(* IEC 61131-3 sources: F100R_S278_Temperville/MyController.device.xml.v3^/Plc Logic.plclogic.xml.v3^/Application.application.xml.v3^/02_Operação (part 4) *)

(* ---- P_ComandosEventos.prg.st ---- *)
PROGRAM P_ComandosEventos
VAR
	TonInicioCicloEventos: ton;
	TonInicioCicloEventosIn: BOOL;
	TonInicioCicloEventosQ: BOOL;
	///------------ Disjuntores ----------------
	TpDisjGeralOn: PulsoPositivo;
	TpDisjGeralOff: PulsoPositivo;
	TpDisjResistOn: PulsoPositivo;
	TpDisjResistOff: PulsoPositivo;
	///------- Comandos Mesa de Operação -------
	TpOperacaoStandby: PulsoPositivo;
	TpOperacaoHabilitada: PulsoPositivo;
	TpBtEmergencia09On: PulsoPositivo;
	TpBtEmergencia09Off: PulsoNegativo;
	TpBt01ResetEmergencia: PulsoPositivo;
	///--- Comandos Mesa de Operação Manual ---
	TpOperacaoManual: PulsoPositivo;
	TpOperacaoAutoma: PulsoPositivo;
	TpBtEmergencia10On: PulsoPositivo;
	TpBtEmergencia10Off: PulsoNegativo;
	TpBt02ResetEmergencia: PulsoPositivo;
	///------ Comandos Mesa de Entrada ------
	TpBtEmergencia01On: PulsoPositivo;
	TpBtEmergencia01Off: PulsoNegativo;
	TpBtEmergencia02On: PulsoPositivo;
	TpBtEmergencia02Off: PulsoNegativo;
	TpBtConfirmaCarga: PulsoPositivo;
	TpChAvancoMeEntOn: PulsoPositivo;
	TpChAvancoMeEntOff: PulsoNegativo;
	TpChRecuoMeEntOn: PulsoPositivo;
	TpChRecuoMeEntOff: PulsoNegativo;
	TpGradeEntradaUp: PulsoPositivo;
	TpGradeEntradaDown: PulsoNegativo;
	TpBtEmergencia03On: PulsoPositivo;
	TpBtEmergencia03Off: PulsoNegativo;
	TpBtEmergencia04On: PulsoPositivo;
	TpBtEmergencia04Off: PulsoNegativo;
	///------ Comandos do Resfriamento ------
	TpBtEmergencia05On: PulsoPositivo;
	TpBtEmergencia05Off: PulsoNegativo;
	TpChAbreResfSup01: PulsoPositivo;
	TpChFechaResfSup01: PulsoNegativo;
	TpChAbreResfInf01: PulsoPositivo;
	TpChFechaResfInf01: PulsoNegativo;
	TpChAbreResfSup02: PulsoPositivo;
	TpChFechaResfSup02: PulsoNegativo;
	TpChAbreResfInf02: PulsoPositivo;
	TpChFechaResfInf02: PulsoNegativo;
	TpBtEmergencia06On: PulsoPositivo;
	TpBtEmergencia06Off: PulsoNegativo;
	TpChAvancoLimpVidroOn: PulsoPositivo;
	TpChAvancoLimpVidroOff: PulsoNegativo;
	TpChRecuoLimpVidroOn: PulsoPositivo;
	TpChRecuoLimpVidroOff: PulsoNegativo;
	///------- Comandos Mesa de Saida -------
	TpBtEmergencia07On: PulsoPositivo;
	TpBtEmergencia07Off: PulsoNegativo;
	TpChAvancoMeSaiOn: PulsoPositivo;
	TpChAvancoMeSaiOff: PulsoNegativo;
	TpChRecuoMeSaiOn: PulsoPositivo;
	TpChRecuoMeSaiOff: PulsoNegativo;
	TpGradeSaidaUp: PulsoPositivo;
	TpGradeSaidaDown: PulsoNegativo;
	TpBtEmergencia08On: PulsoPositivo;
	TpBtEmergencia08Off: PulsoNegativo;
	///------ Comandos do Supervisório ------
	TpBtEnvioDeReceita: PulsoPositivo;
	TpBtHmiIniciaCiclo: PulsoPositivo;
	TpBtHmiFinalizaCiclo: PulsoPositivo;
	TpBtSairForno: PulsoPositivo;
	TpBtSairResfriamento: PulsoPositivo;
	TpBtAbrePortaEntrForno: PulsoPositivo;
	TpBtFechaPortaEntForno: PulsoNegativo;
	TpBtAbrePortaSaidaForno: PulsoPositivo;
	TpBtFechaPortaSaidForno: PulsoNegativo;
	TpBtForceConveccaoOn: PulsoPositivo;
	TpBtForceConveccaoOff: PulsoNegativo;
	TpBtSobeForno: PulsoPositivo;
	TpBtDesceForno: PulsoPositivo;
	TpTesteAutoResistencia: PulsoPositivo;
	TpTesteAutoResistFim: PulsoPositivo;
	TpTesteAutoResistAbort: PulsoPositivo;
	TpProgrHorariaAtivada: PulsoPositivo;
	TpProgrHorariaDesativada: PulsoNegativo;
	TpProgrHorariaIniciadda: PulsoPositivo;
	TpBtLigaAquecimentoRampa: PulsoPositivo;
	TpBtLigaAquecimento: PulsoPositivo;
	TpBtDesligaAquecimento: PulsoPositivo;
	TpResistenciaLigada: PulsoPositivo;
	TpResistenciaDesligada: PulsoNegativo;
	TpHomeDutosIniciado: PulsoPositivo;
	TpHomeDutosOK: PulsoPositivo;
	TpHomeGuilhotinaIniciado: PulsoPositivo;
	TpHomeGuilhotinaOK: PulsoPositivo;
END_VAR

//Registro de Eventos

//Sinais Retorno Disjuntores
(*----------- Disjuntor Geral -------------*)
TpDisjGeralOn	(Entrada:= xDisjGeralOn, 	SaidaPulsoPo=> );
TpDisjGeralOff	(Entrada:= xDisjGeralOff, 	SaidaPulsoPo=> );

(*-------- Disjuntor Resistências ---------*)
TpDisjResistOn	(Entrada:= xDisjResistOn, 	SaidaPulsoPo=> );
TpDisjResistOff	(Entrada:= xDisjResistOff, 	SaidaPulsoPo=> );

//Sinais de Acionamento de Botoes Fisicos
(*------- Comandos Mesa de Operação -------*)
TpOperacaoHabilitada	(Entrada:= xOperacaoHabilitada, 	SaidaPulsoPo=> );
TpOperacaoStandby		(Entrada:= xOperacaoStandBy, 		SaidaPulsoPo=> );
TpBtEmergencia09On		(Entrada:= xBt09Emergencia, 		SaidaPulsoPo=> );
TpBtEmergencia09Off		(Entrada:= xBt09Emergencia, 		SaidaPulsoNe=> );
TpBt01ResetEmergencia	(Entrada:= xBt01CalaAlarme, 		SaidaPulsoPo=> );

(*--- Comandos Mesa de Operação Manual ---*)
TpOperacaoManual		(Entrada:= xOperacaoManual, 		SaidaPulsoPo=> );
TpOperacaoAutoma		(Entrada:= xOperacaoAutoma, 		SaidaPulsoPo=> );
TpBtEmergencia10On		(Entrada:= xBt10Emergencia,			SaidaPulsoPo=> );
TpBtEmergencia10Off		(Entrada:= xBt10Emergencia,			SaidaPulsoNe=> );
TpBt02ResetEmergencia	(Entrada:= xBt02CalaAlarme, 		SaidaPulsoPo=> );

(*------ Comandos Mesa de Entrada ------*)
TpBtEmergencia01On		(Entrada:= xBt01Emergencia,			SaidaPulsoPo=> );
TpBtEmergencia01Off		(Entrada:= xBt01Emergencia,			SaidaPulsoNe=> );
TpBtEmergencia02On		(Entrada:= xBt02Emergencia,			SaidaPulsoPo=> );
TpBtEmergencia02Off		(Entrada:= xBt02Emergencia,			SaidaPulsoNe=> );
TpBtConfirmaCarga		(Entrada:= xBtHabilitaCarregamento,	SaidaPulsoPo=> );
TpChAvancoMeEntOn		(Entrada:= xChAvancaMesaEntrada,	SaidaPulsoPo=> );
TpChAvancoMeEntOff		(Entrada:= xChAvancaMesaEntrada,	SaidaPulsoNe=> );
TpChRecuoMeEntOn		(Entrada:= xChRecuaMesaEntrada,		SaidaPulsoPo=> );
TpChRecuoMeEntOff		(Entrada:= xChRecuaMesaEntrada,		SaidaPulsoNe=> );
TpGradeEntradaUp		(Entrada:= xValvulaGradeEntrada,	SaidaPulsoPo=> );
TpGradeEntradaDown		(Entrada:= xValvulaGradeEntrada,	SaidaPulsoNe=> );
TpBtEmergencia03On		(Entrada:= xBt03Emergencia,			SaidaPulsoPo=> );
TpBtEmergencia03Off		(Entrada:= xBt03Emergencia,			SaidaPulsoNe=> );
TpBtEmergencia04On		(Entrada:= xBt04Emergencia,			SaidaPulsoPo=> );
TpBtEmergencia04Off		(Entrada:= xBt04Emergencia,			SaidaPulsoNe=> );

(*------ Comandos do Resfriamento ------*)
TpBtEmergencia05On		(Entrada:= xBt05Emergencia,			SaidaPulsoPo=> );
TpBtEmergencia05Off		(Entrada:= xBt05Emergencia,			SaidaPulsoNe=> );
TpChAbreResfSup01		(Entrada:= xChAbreDuctosResfriadorSup01,SaidaPulsoPo=> );
TpChFechaResfSup01		(Entrada:= xChAbreDuctosResfriadorSup01,SaidaPulsoNe=> );
TpChAbreResfInf01		(Entrada:= xChAbreDuctosResfriadorInf01,SaidaPulsoPo=> );
TpChFechaResfInf01		(Entrada:= xChAbreDuctosResfriadorInf01,SaidaPulsoNe=> );
TpChAbreResfSup02		(Entrada:= xChAbreDuctosResfriadorSup02,SaidaPulsoPo=> );
TpChFechaResfSup02		(Entrada:= xChAbreDuctosResfriadorSup02,SaidaPulsoNe=> );
TpChAbreResfInf02		(Entrada:= xChAbreDuctosResfriadorInf02,SaidaPulsoPo=> );
TpChFechaResfInf02		(Entrada:= xChAbreDuctosResfriadorInf02,SaidaPulsoNe=> );
TpBtEmergencia06On		(Entrada:= xBt06Emergencia,				SaidaPulsoPo=> );
TpBtEmergencia06Off		(Entrada:= xBt06Emergencia,				SaidaPulsoNe=> );
TpChAvancoLimpVidroOn	(Entrada:= xChAvancoLimpaResfriador02,	SaidaPulsoPo=> );
TpChAvancoLimpVidroOff	(Entrada:= xChAvancoLimpaResfriador02,	SaidaPulsoNe=> );
TpChRecuoLimpVidroOn	(Entrada:= xChRecuoLimpaResfriador02,	SaidaPulsoPo=> );
TpChRecuoLimpVidroOff	(Entrada:= xChRecuoLimpaResfriador02,	SaidaPulsoNe=> );

(*------- Comandos Mesa de Saida -------*)
TpBtEmergencia07On		(Entrada:= xBt07Emergencia,		SaidaPulsoPo=> );
TpBtEmergencia07Off		(Entrada:= xBt07Emergencia,		SaidaPulsoNe=> );
TpChAvancoMeSaiOn		(Entrada:= xChAvancaMesaSaida,	SaidaPulsoPo=> );
TpChAvancoMeSaiOff		(Entrada:= xChAvancaMesaSaida,	SaidaPulsoNe=> );
TpChRecuoMeSaiOn		(Entrada:= xChRecuaMesaSaida,	SaidaPulsoPo=> );
TpChRecuoMeSaiOff		(Entrada:= xChRecuaMesaSaida,	SaidaPulsoNe=> );
TpGradeSaidaUp			(Entrada:= xValvulaGradeSaida,	SaidaPulsoPo=> );
TpGradeSaidaDown		(Entrada:= xValvulaGradeSaida,	SaidaPulsoNe=> );
TpBtEmergencia08On		(Entrada:= xBt08Emergencia,		SaidaPulsoPo=> );
TpBtEmergencia08Off		(Entrada:= xBt08Emergencia,		SaidaPulsoNe=> );

//Sinais de Acionamento de Botoes Logicos

TpBtEnvioDeReceita		(Entrada:= xReceitaEnviadaEventos,	SaidaPulsoPo=> );
xReceitaEnviadaEventos:=FALSE;
TpBtHmiIniciaCiclo		(Entrada:= xBtHmiIniciaCiclo, 		SaidaPulsoPo=> );
TpBtHmiFinalizaCiclo	(Entrada:= xBtHmiFinalizaCiclo, 	SaidaPulsoPo=> );
TpBtSairForno			(Entrada:= xSairForno, 			SaidaPulsoPo=> );
TpBtSairResfriamento	(Entrada:= xSairResfriamentoEventos,SaidaPulsoPo=> );
xSairResfriamentoEventos:=FALSE;
TpBtAbrePortaEntrForno	(Entrada:= xPortaEntradaFornoForce, SaidaPulsoPo=> );
TpBtFechaPortaEntForno	(Entrada:= xPortaEntradaFornoForce, SaidaPulsoNe=> );
TpBtAbrePortaSaidaForno	(Entrada:= xPortaSaidaFornoForce, 	SaidaPulsoPo=> );
TpBtFechaPortaSaidForno	(Entrada:= xPortaSaidaFornoForce, 	SaidaPulsoNe=> );
TpBtForceConveccaoOn	(Entrada:= xForceConveccao, 		SaidaPulsoPo=> );
TpBtForceConveccaoOff	(Entrada:= xForceConveccao, 		SaidaPulsoNe=> );
TpBtSobeForno			(Entrada:= xBtSobeForno	, 			SaidaPulsoPo=> );
TpBtDesceForno			(Entrada:= xBtDesceForno,		 	SaidaPulsoPo=> );
TpTesteAutoResistencia	(Entrada:= bIniciaTesteResistencias,SaidaPulsoPo=> );
TpTesteAutoResistAbort	(Entrada:= bAbortaTesteResistencias,SaidaPulsoPo=> );
TpTesteAutoResistFim	(Entrada:= bResetTesteResistencias,	SaidaPulsoPo=> );
TpProgrHorariaAtivada	(Entrada:= xStatusAtvProgHoraria, 	SaidaPulsoPo=> );
TpProgrHorariaDesativada(Entrada:= xStatusAtvProgHoraria, 	SaidaPulsoNe=> );
TpProgrHorariaIniciadda	(Entrada:= xDataHoraProgOk, 		SaidaPulsoPo=> );

TpBtLigaAquecimentoRampa(Entrada:= xBtLigaResRampa, 	SaidaPulsoPo=> );
xBtLigaResRampa:=FALSE;
TpBtLigaAquecimento		(Entrada:= xBtLigaResCiclo, 	SaidaPulsoPo=> );
xBtLigaResCiclo:=FALSE;
TpBtDesligaAquecimento	(Entrada:= xBtDeslResCiclo, 	SaidaPulsoPo=> );
xBtDeslResCiclo:=FALSE;

TpResistenciaLigada		(Entrada:= xResistenciasLigadas, 	SaidaPulsoPo=> );
TpResistenciaDesligada	(Entrada:= xResistenciasLigadas, 	SaidaPulsoNe=> );

TpHomeDutosIniciado		(Entrada:= , 	SaidaPulsoPo=> );
TpHomeDutosOK			(Entrada:=xHomeDuctosResfriadorSup01Ok , 	SaidaPulsoPo=> );
TpHomeGuilhotinaIniciado(Entrada:= , 	SaidaPulsoPo=> );
TpHomeGuilhotinaOK		(Entrada:=xHomeGuilhotina01Ok , 	SaidaPulsoPo=> );

// Tempo para Inicio de Ciclo

TonInicioCicloEventosIn:=TRUE;
TonInicioCicloEventos(IN:=TonInicioCicloEventosIn , PT:=T#200MS , Q=>TonInicioCicloEventosQ, ET=> );

IF TonInicioCicloEventosQ THEN

	(*------------- Disjuntores ---------------*)
	IF TpDisjGeralOn.SaidaPulsoPo			THEN bDisjGeralOn	:=TRUE;		END_IF;
	IF TpDisjGeralOff.SaidaPulsoPo			THEN bDisjGeralOff	:=TRUE;		END_IF;
	IF TpDisjResistOn.SaidaPulsoPo			THEN bDisjResistOn	:=TRUE;		END_IF;
	IF TpDisjResistOff.SaidaPulsoPo			THEN bDisjResistOff	:=TRUE;		END_IF;

	(*------- Comandos Mesa de Operação -------*)
	IF TpOperacaoStandby.SaidaPulsoPo 		THEN bMaquinaOperacaoStandby:=TRUE;		END_IF;
	IF TpOperacaoHabilitada.SaidaPulsoPo 	THEN bMaquinaOperacaoHabilitada:=TRUE;	END_IF;
	IF TpBtEmergencia01On.SaidaPulsoPo 		THEN bEmergencia01On:=TRUE;		END_IF;
	IF TpBtEmergencia01Off.SaidaPulsoNe 	THEN bEmergencia01Off:=TRUE;	END_IF;
	IF TpBt01ResetEmergencia.SaidaPulsoPo	THEN b01ResetEmergencia:=TRUE;  END_IF;

	(*--- Comandos Mesa de Operação Manual ---*)
	IF TpOperacaoManual.SaidaPulsoPo 		THEN bMaquinaEmManual:=TRUE;		END_IF;
	IF TpOperacaoAutoma.SaidaPulsoPo 		THEN bMaquinaEmAutoma:=TRUE;		END_IF;
	IF TpBtEmergencia10On.SaidaPulsoPo 		THEN bEmergencia10On:=TRUE;		END_IF;
	IF TpBtEmergencia10Off.SaidaPulsoNe 	THEN bEmergencia10Off:=TRUE;	END_IF;
	IF TpBt02ResetEmergencia.SaidaPulsoPo	THEN b02ResetEmergencia:=TRUE;  END_IF;

	(*------ Comandos Mesa de Entrada ------*)
	IF TpBtEmergencia02On.SaidaPulsoPo 		THEN bEmergencia02On:=TRUE;		END_IF;
	IF TpBtEmergencia02Off.SaidaPulsoNe 	THEN bEmergencia02Off:=TRUE;	END_IF;
	IF TpBtConfirmaCarga.SaidaPulsoPo 		THEN bConfirmaCarga:=TRUE;		END_IF;
	IF TpChAvancoMeEntOn.SaidaPulsoPo 		THEN bAvancoMeEntOn:=TRUE;		END_IF;
	IF TpChAvancoMeEntOff.SaidaPulsoNe 		THEN bAvancoMeEntOff:=TRUE;		END_IF;
	IF TpChRecuoMeEntOn.SaidaPulsoPo 		THEN bRecuoMeEntOn:=TRUE;		END_IF;
	IF TpChRecuoMeEntOff.SaidaPulsoNe 		THEN bRecuoMeEntOff:=TRUE;		END_IF;
	IF TpGradeEntradaUp.SaidaPulsoPo 		THEN bGradeEntradaUp:=TRUE;		END_IF;
	IF TpGradeEntradaDown.SaidaPulsoNe 		THEN bGradeEntradaDown:=TRUE;	END_IF;

	(*------ Comandos do Resfriamento ------*)
	IF TpBtEmergencia03On.SaidaPulsoPo 		THEN bEmergencia03On:=TRUE;		END_IF;
	IF TpBtEmergencia03Off.SaidaPulsoNe 	THEN bEmergencia03Off:=TRUE;	END_IF;
	IF TpBtEmergencia05On.SaidaPulsoPo 		THEN bEmergencia05On:=TRUE;		END_IF;
	IF TpBtEmergencia05Off.SaidaPulsoNe 	THEN bEmergencia05Off:=TRUE;	END_IF;
	IF TpChAbreResfSup01.SaidaPulsoPo 		THEN bAbreResfSup01:=TRUE;		END_IF;
	IF TpChFechaResfSup01.SaidaPulsoNe 		THEN bFechaResfSup01:=TRUE;		END_IF;
	IF TpChAbreResfInf01.SaidaPulsoPo 		THEN bAbreResfInf01:=TRUE;		END_IF;
	IF TpChFechaResfInf01.SaidaPulsoNe 		THEN bFechaResfInf01:=TRUE;		END_IF;
	IF TpChAbreResfSup02.SaidaPulsoPo 		THEN bAbreResfSup02:=TRUE;		END_IF;
	IF TpChFechaResfSup02.SaidaPulsoNe 		THEN bFechaResfSup02:=TRUE;		END_IF;
	IF TpChAbreResfInf02.SaidaPulsoPo 		THEN bAbreResfInf02:=TRUE;		END_IF;
	IF TpChFechaResfInf02.SaidaPulsoNe 		THEN bFechaResfInf02:=TRUE;		END_IF;
	IF TpBtEmergencia06On.SaidaPulsoPo 		THEN bEmergencia06On:=TRUE;		END_IF;
	IF TpBtEmergencia06Off.SaidaPulsoNe 	THEN bEmergencia06Off:=TRUE;	END_IF;
	IF TpChAvancoLimpVidroOn.SaidaPulsoPo 	THEN bAvancoLimpVidroOn:=TRUE;	END_IF;
	IF TpChAvancoLimpVidroOff.SaidaPulsoNe 	THEN bAvancoLimpVidroOff:=TRUE;	END_IF;
	IF TpChRecuoLimpVidroOn.SaidaPulsoPo 	THEN bRecuoLimpVidroOn:=TRUE;	END_IF;
	IF TpChRecuoLimpVidroOff.SaidaPulsoNe 	THEN bRecuoLimpVidroOff:=TRUE;	END_IF;

	(*------- Comandos Mesa de Saida -------*)
	IF TpBtEmergencia04On.SaidaPulsoPo 		THEN bEmergencia04On:=TRUE;		END_IF;
	IF TpBtEmergencia04Off.SaidaPulsoNe 	THEN bEmergencia04Off:=TRUE;	END_IF;
	IF TpBtEmergencia07On.SaidaPulsoPo 		THEN bEmergencia07On:=TRUE;		END_IF;
	IF TpBtEmergencia07Off.SaidaPulsoNe 	THEN bEmergencia07Off:=TRUE;	END_IF;
	IF TpChAvancoMeSaiOn.SaidaPulsoPo 		THEN bAvancoMeSaiOn:=TRUE;		END_IF;
	IF TpChAvancoMeSaiOff.SaidaPulsoNe 		THEN bAvancoMeSaiOff:=TRUE;		END_IF;
	IF TpChRecuoMeSaiOn.SaidaPulsoPo 		THEN bRecuoMeSaiOn:=TRUE;		END_IF;
	IF TpChRecuoMeSaiOff.SaidaPulsoNe 		THEN bRecuoMeSaiOff:=TRUE;		END_IF;
	IF TpGradeSaidaUp.SaidaPulsoPo 			THEN bGradeSaidaUp:=TRUE;		END_IF;
	IF TpGradeSaidaDown.SaidaPulsoNe 		THEN bGradeSaidaDown:=TRUE;		END_IF;
	IF TpBtEmergencia08On.SaidaPulsoPo 		THEN bEmergencia08On:=TRUE;		END_IF;
	IF TpBtEmergencia08Off.SaidaPulsoNe 	THEN bEmergencia08Off:=TRUE;	END_IF;

	(*------ Comandos do Supervisório ------*)
	IF TpBtEnvioDeReceita.SaidaPulsoPo 		THEN bEnvioDeReceita:=TRUE; 		END_IF;
	IF TpBtHmiIniciaCiclo.SaidaPulsoPo 		THEN bHimIniciaCiclo:=TRUE; 		END_IF;
	IF TpBtHmiFinalizaCiclo.SaidaPulsoPo 	THEN bHimFinalCiclo:=TRUE; 			END_IF;
	IF TpBtSairForno.SaidaPulsoPo 			THEN bBtSairForno:=TRUE; 			END_IF;
	IF TpBtSairResfriamento.SaidaPulsoPo 	THEN bBtSairResfriamento:=TRUE; 	END_IF;
	IF TpBtAbrePortaEntrForno.SaidaPulsoPo 	THEN bBtAbrePortaEntrForno:=TRUE; 	END_IF;
	IF TpBtFechaPortaEntForno.SaidaPulsoNe 	THEN bBtFechaPortaEntForno:=TRUE; 	END_IF;
	IF TpBtAbrePortaSaidaForno.SaidaPulsoPo	THEN bBtAbrePortaSaidaForno:=TRUE;	END_IF;
	IF TpBtFechaPortaSaidForno.SaidaPulsoNe	THEN bBtFechaPortaSaidForno:=TRUE;	END_IF;
	IF TpBtForceConveccaoOn.SaidaPulsoPo		THEN	bBtForceConveccaoOn:=TRUE;		END_IF;
	IF TpBtForceConveccaoOff.SaidaPulsoNe		THEN	bBtForceConveccaoOff:=TRUE;		END_IF;
	IF TpBtSobeForno.SaidaPulsoPo				THEN	bBtSobeForno:=TRUE;				END_IF;
	IF TpBtDesceForno.SaidaPulsoPo				THEN	bBtDesceForno:=TRUE;			END_IF;
	IF TpTesteAutoResistencia.SaidaPulsoPo		THEN	bTesteAutoResistencia:=TRUE;	END_IF;
	IF TpTesteAutoResistAbort.SaidaPulsoPo		THEN	bTesteAutoResistAbort:=TRUE;	END_IF;
	IF TpTesteAutoResistFim.SaidaPulsoPo		THEN	bTesteAutoResistFim:=TRUE;		END_IF;
	IF TpProgrHorariaAtivada.SaidaPulsoPo		THEN	bProgrHorariaAtivada:=TRUE;		END_IF;
	IF TpProgrHorariaDesativada.SaidaPulsoNe	THEN	bProgrHorariaDesativada:=TRUE;	END_IF;
	IF TpProgrHorariaIniciadda.SaidaPulsoPo		THEN	bProgrHorariaIniciadda:=TRUE;	END_IF;
	IF TpBtLigaAquecimentoRampa.SaidaPulsoPo	THEN	bBtLigaAquecimentoRampa:=TRUE;	END_IF;
	IF TpBtLigaAquecimento.SaidaPulsoPo			THEN	bBtLigaAquecimento:=TRUE;		END_IF;
	IF TpBtDesligaAquecimento.SaidaPulsoPo		THEN	bBtDesligaAquecimento:=TRUE;	END_IF;
	IF TpResistenciaLigada.SaidaPulsoPo			THEN	bResistenciaLigada:=TRUE;		END_IF;
	IF TpResistenciaDesligada.SaidaPulsoNe		THEN	bResistenciaDesligada:=TRUE;	END_IF;

	IF TpHomeDutosIniciado.SaidaPulsoPo			THEN	bHomeDutosIniciado:=TRUE;		END_IF;
	IF TpHomeDutosOK.SaidaPulsoPo				THEN	bHomeDutosOK:=TRUE;				END_IF;
	IF TpHomeGuilhotinaIniciado.SaidaPulsoPo	THEN	bHomeGuilhotinaIniciado:=TRUE;	END_IF;
	IF TpHomeGuilhotinaOK.SaidaPulsoPo			THEN	bHomeGuilhotinaOK:=TRUE;		END_IF;

END_IF

(* ---- Q_Conveccao.prg.st ---- *)
PROGRAM Q_Conveccao
VAR
	TemporizadorConveccao: TON;
	TemporizadorConveccaoIn: BOOL;
	TemporizadorConveccaoEt: TIME;
	TempoConveccaoOnOff: TimerGeneration;
	TempoConveccaoOnOffEnable: BOOL;
	TempoConveccaoOnOffTimeLow: TIME;
	TempoConveccaoOnOffTimeHigh: TIME;
	TempoConveccaoOnOffOut: BOOL;
	ForceConveccao: HabilitaDesabilita;
	xAcionaConveccaoAuto: BOOL;
END_VAR

(*----------- SISTEMA DE CONVECÇÃO --------------------*)

// Funcionamento em Automático

//Habilita/Desabilita
xConveccaoHabilitado:= iTempoConveccao<>0 and iTempoConveccaoAberta<>0;

//Liga
IF xConveccaoHabilitado AND xLigaConveccaoForno THEN
	xAcionaConveccaoAuto:=TRUE;
	xLigaConveccaoForno:=FALSE;
END_IF

//Temporiza
TemporizadorConveccaoIn:=xAcionaConveccaoAuto;
TemporizadorConveccao(IN:=TemporizadorConveccaoIn , PT:=t#999s , Q=> , ET=>TemporizadorConveccaoEt );

//Tempo de Convecção decorrido
iTempoConveccaoDecorrido:=DINT_TO_INT(TIME_TO_DINT(TemporizadorConveccaoEt)/1000);

//Compara
IF (iTempoConveccaoDecorrido>=iTempoConveccao) OR NOT xConveccaoHabilitado OR xOperacaoManual THEN
	xAcionaConveccaoAuto:=FALSE;
END_IF

// Force em Manual

ForceConveccao(
	Entrada:= xBtForceConveccao,
	Entrada02:= ,
	Entrada03:= xOperacaoManual,
	Alarme01:= ,
	Alarme02:= ,
	Alarme03:= ,
	StatusSaida=> xForceConveccao);

IF xBtForceConveccao THEN
	xBtForceConveccao:=FALSE;
END_IF

TempoConveccaoOnOffTimeLow:= DINT_TO_TIME(INT_TO_DINT(iTempoConveccaoAberta)*1000);
TempoConveccaoOnOffTimeHigh:= DINT_TO_TIME(INT_TO_DINT(iTempoConveccaoFechada)*1000);
TempoConveccaoOnOffEnable:=xAcionaConveccaoAuto OR xForceConveccao;
TempoConveccaoOnOff(ENABLE:=TempoConveccaoOnOffEnable , TIMELOW:=TempoConveccaoOnOffTimeLow , TIMEHIGH:=TempoConveccaoOnOffTimeHigh , OUT=>TempoConveccaoOnOffOut );

xValvulaConveccao:=TempoConveccaoOnOffOut;
xValvulaConveccaoLigada:=xValvulaConveccao OR xForceConveccao;

IF xOperacaoManual THEN
	xLigaConveccaoForno:=FALSE;
	xAcionaConveccaoAuto:=FALSE;
END_IF

(* ---- R_ManometroDifusor.prg.st ---- *)
PROGRAM R_ManometroDifusor
VAR
	MediaValoresDifusor01: RegistradorMedia;
	MediaValoresDifusor02: RegistradorMedia;
	rValorLeituraPressaoDifusor01: REAL;
	rValorLeituraPressaoAuxiliarDif01: REAL;
	rValorLeituraPressaoDifusor02: REAL;
	rValorLeituraPressaoAuxiliarDif02: REAL;
END_VAR

// ----------------------Manometro Difusor 01------------------------------

MediaValoresDifusor01.rDadoEntrada:=INT_TO_REAL(iValorLeituraPressaoDifusor01);

MediaValoresDifusor01(rDadoEntrada:= , rDadoSaida=>rValorLeituraPressaoAuxiliarDif01 );

IF	rValorLeituraPressaoAuxiliarDif01<= 200 THEN
	rValorLeituraPressaoDifusor01:=0;
ELSE
	rValorLeituraPressaoDifusor01:=rValorLeituraPressaoAuxiliarDif01;
END_IF

rValorLeituraPressaoDifusor01Mbar:= 1000*rValorLeituraPressaoDifusor01/32767;
rValorLeituraPressaoDifusor01Bar:=rValorLeituraPressaoDifusor01Mbar/1000;
rValorLeituraPressaoDifusor01Psi:=rValorLeituraPressaoDifusor01Bar/0.068948;

rValorLeituraPressaoDifusor01InHg:=rValorLeituraPressaoDifusor01Bar*29.5299889;
rValorLeituraPressaoDifusor01CmHg:=rValorLeituraPressaoDifusor01Bar*75.006375;
rValorLeituraPressaoDifusor01MmHg:=rValorLeituraPressaoDifusor01Bar*750.06375;
rValorLeituraPressaoDifusor01MmCa:=rValorLeituraPressaoDifusor01Bar*10197.1621;

// ----------------------Manometro Difusor 02------------------------------

MediaValoresDifusor02.rDadoEntrada:=INT_TO_REAL(iValorLeituraPressaoDifusor02);

MediaValoresDifusor02(rDadoEntrada:= , rDadoSaida=>rValorLeituraPressaoAuxiliarDif02 );

IF	rValorLeituraPressaoAuxiliarDif02<= 200 THEN
	rValorLeituraPressaoDifusor02:=0;
ELSE
	rValorLeituraPressaoDifusor02:=rValorLeituraPressaoAuxiliarDif02;
END_IF

rValorLeituraPressaoDifusor02Mbar:= 1000*rValorLeituraPressaoDifusor02/32767;
rValorLeituraPressaoDifusor02Bar:=rValorLeituraPressaoDifusor02Mbar/1000;
rValorLeituraPressaoDifusor02Psi:=rValorLeituraPressaoDifusor02Bar/0.068948;

rValorLeituraPressaoDifusor02InHg:=rValorLeituraPressaoDifusor02Bar*29.5299889;
rValorLeituraPressaoDifusor02CmHg:=rValorLeituraPressaoDifusor02Bar*75.006375;
rValorLeituraPressaoDifusor02MmHg:=rValorLeituraPressaoDifusor02Bar*750.06375;
rValorLeituraPressaoDifusor02MmCa:=rValorLeituraPressaoDifusor02Bar*10197.1621;

(* ---- R_Pressostato.prg.st ---- *)
PROGRAM R_Pressostato
VAR
	TonPressBaixaRede: TON;
	TonPressAltaRede: TON;
	TpAlmRedeSom: TP;
	TpAlmRedeSomIn: BOOL;
	TonPressBaixaMaq: TON;
	TonPressAltaMaq: TON;
	TpAlmMaqSom: TP;
	AlarmePressaoArAltaRede: BOOL;
	AlarmePressaoArBaixaRede: BOOL;
	AlarmePressaoArMaqAlta: BOOL;
	AlarmePressaoArMaqBaixa: BOOL;
END_VAR

// PRESSOSTATO DA REDE DE ALIMENTAÇÃO DE AR COMPRIMIDO
(*-----------(* OPÇÃO COM DUAS SAIDAS DIGITAIS *)-------------*)
// Status da Pressão de Ar na Rede
IF NOT xPressaoBaixaMediaRede AND NOT xPressaoMediaAltaRede THEN
	iPressaoDaRede:=0; // Baixa
END_IF

IF xPressaoBaixaMediaRede AND NOT xPressaoMediaAltaRede THEN
	iPressaoDaRede:=1; // Normal
END_IF

IF xPressaoBaixaMediaRede AND xPressaoMediaAltaRede THEN
	iPressaoDaRede:=2; // Alta
END_IF

// Alarmes
IF iPressaoDaRede<=0 AND NOT xValvulaConveccaoLigada THEN (* Pressão baixa *)
	AlarmePressaoArBaixaRede:=TRUE; (* alarme de pressão baixa *)
ELSE
	AlarmePressaoArBaixaRede:=FALSE;
END_IF

IF iPressaoDaRede>=2 THEN (* Pressão alta *)
	AlarmePressaoArAltaRede:=TRUE; (* alarme de pressão alta *)
ELSE
	AlarmePressaoArAltaRede:=FALSE;
END_IF

TonPressBaixaRede.IN:= AlarmePressaoArBaixaRede;
TonPressAltaRede.IN:= AlarmePressaoArAltaRede;

TonPressBaixaRede(PT:=T#1000MS );
TonPressAltaRede(PT:=T#1000MS );

IF TonPressBaixaRede.Q THEN
	xAlarmePressaoArBaixaRede:= TRUE;
END_IF

IF TonPressAltaRede.Q THEN
	xAlarmePressaoArAltaRede:=TRUE;
END_IF

xAlarmePressaoArRede:= xAlarmePressaoArBaixaRede OR xAlarmePressaoArAltaRede;

TpAlmRedeSomIn:= xAlarmePressaoArRede AND xMaquinaEmCiclo;

//Sinais de Alarme
TpAlmRedeSom(IN:= TpAlmRedeSomIn, PT:= T#500MS );

IF TpAlmRedeSom.Q THEN
	xAlarmePressaoArRedeSom:=TRUE;
END_IF

IF	bResetAlmGeral THEN
	xAlarmePressaoArBaixaRede:=FALSE;
	xAlarmePressaoArAltaRede:=FALSE;
	xAlarmePressaoArRedeSom:=FALSE;
END_IF

////////////////////////////////////////////////////////////////////////
// PRESSOSTATO DA REDE DE ALIMENTAÇÃO DE AR COMPRIMIDO
(*-----------(* OPÇÃO COM UMA SAIDAS DIGITAIS *)-------------*)
// Status da Pressão de Ar na Rede
(*IF NOT xPressaoBaixaMedia THEN
	iPressaoDaRede:=0; // Baixa
END_IF

IF xPressaoBaixaMedia THEN
	iPressaoDaRede:=1; // Normal
END_IF

// Alarmes
IF iPressaoDaRede<=0 AND NOT xValvulaConveccaoLigada THEN (* Pressão baixa *)
	AlarmePressaoArBaixa:=TRUE; (* alarme de pressão baixa *)
ELSE
	AlarmePressaoArBaixa:=FALSE;
END_IF

TonPressBaixaRede.IN:= AlarmePressaoArBaixa;

TonPressBaixaRede(PT:=T#1000MS );

IF TonPressBaixaRede.Q THEN
	xAlarmePressaoArBaixaRede:= TRUE;
END_IF

xAlarmePressaoArRede:= xAlarmePressaoArBaixaRede OR xAlarmePressaoArAltaRede;

//Sinais de Alarme
TpAlmRedeSom(IN:= xAlarmePressaoArRede, PT:= T#500MS );

IF TpAlmRedeSom.Q THEN
	xAlarmePressaoArRedeSom:=TRUE;
END_IF

IF	bResetAlmGeral THEN
	xAlarmePressaoArBaixaRede:=FALSE;
	xAlarmePressaoArAltaRede:=FALSE;
	xAlarmePressaoArRedeSom:=FALSE;
END_IF
*)
////////////////////////////////////////////////////////////////////
//PRESSOSTATO DA ENTRADA DA MÁQUINA
(*-----------(* OPÇÃO COM SAIDAS ANALÓGICA *)-------------*)
// Status da Pressão de Ar na Rede
(*IF rValorPressaoMaqBar < 5.0 THEN
	iPressaoDaMaquina:=0; // Baixa
END_IF

IF rValorPressaoMaqBar >= 5.0 AND rValorPressaoMaqBar <= 7.0 THEN
	iPressaoDaMaquina:=1; // Normal
END_IF

IF rValorPressaoMaqBar > 7.0 THEN
	iPressaoDaMaquina:=2; // Alta
END_IF

// Alarmes
IF iPressaoDaMaquina<=0 AND NOT xValvulaConveccaoLigada THEN (* Pressão baixa *)
	AlarmePressaoArMaqBaixa:=TRUE; (* alarme de pressão baixa *)
ELSE
	AlarmePressaoArMaqBaixa:=FALSE;
END_IF

IF iPressaoDaMaquina>=2 THEN (* Pressão alta *)
	AlarmePressaoArMaqAlta:=TRUE; (* alarme de pressão alta *)
ELSE
	AlarmePressaoArMaqAlta:=FALSE;
END_IF

TonPressBaixaMaq.IN:= AlarmePressaoArMaqBaixa;
TonPressAltaMaq.IN:= AlarmePressaoArMaqAlta;

TonPressBaixaMaq(PT:=T#1000MS );
TonPressAltaMaq(PT:=T#2000MS );

IF TonPressBaixaMaq.Q THEN
	xAlarmePressaoArBaixaMaq:= TRUE;
END_IF

IF TonPressAltaMaq.Q THEN
	xAlarmePressaoArAltaMaq:=TRUE;
END_IF

xAlarmePressaoArMaq:= xAlarmePressaoArBaixaMaq OR xAlarmePressaoArAltaMaq;

//Sinais de Alarme
TpAlmMaqSom(IN:= xAlarmePressaoArMaq, PT:= T#500MS );

IF TpAlmMaqSom.Q THEN
	xAlarmePressaoArMaqSom:=TRUE;
END_IF

IF	bResetAlmGeral THEN
	xAlarmePressaoArBaixaMaq:=FALSE;
	xAlarmePressaoArAltaMaq:=FALSE;
	xAlarmePressaoArMaqSom:=FALSE;
END_IF
*)

(* ---- R_PressostatoAnal.prg.st ---- *)
PROGRAM R_PressostatoAnal
VAR
	MediaValoresPressRede: RegistradorMedia;
	rValorLeituraPressaoRede: REAL;
	MediaValoresPressMaq: RegistradorMedia;
	rValorLeituraPressaoMaq: REAL;
END_VAR

// PRESSOSTATO PRESSÃO DA REDE DE ALIMENTAÇÃO DA MAQUINA
MediaValoresPressRede.rDadoEntrada:=INT_TO_REAL(iValorLeituraPressaoRede);

MediaValoresPressRede(rDadoEntrada:= , rDadoSaida=>rValorLeituraPressaoRede );

rValorPressaoRedeMpa:= rValorLeituraPressaoRede/32767;
rValorPressaoRedeBar:=rValorPressaoRedeMpa*10;
rValorPressaoRedePsi:=rValorPressaoRedeBar/0.068948;

rValorPressaoRedeInHg:=rValorPressaoRedeBar*29.5299889;
rValorPressaoRedeCmHg:=rValorPressaoRedeBar*75.006375;
rValorPressaoRedeMmHg:=rValorPressaoRedeBar*750.06375;
rValorPressaoRedeMmCa:=rValorPressaoRedeBar*10197.1621;

// PRESSOSTATO PRESSÃO DA MAQUINA
MediaValoresPressMaq.rDadoEntrada:=INT_TO_REAL(iValorLeituraPressaoMaq);

MediaValoresPressMaq(rDadoEntrada:= , rDadoSaida=>rValorLeituraPressaoMaq );

rValorPressaoMaqMpa:= rValorLeituraPressaoMaq/32767;
rValorPressaoMaqBar:=rValorPressaoMaqMpa*10;
rValorPressaoMaqPsi:=rValorPressaoMaqBar/0.068948;

rValorPressaoMaqInHg:=rValorPressaoMaqBar*29.5299889;
rValorPressaoMaqCmHg:=rValorPressaoMaqBar*75.006375;
rValorPressaoMaqMmHg:=rValorPressaoMaqBar*750.06375;
rValorPressaoMaqMmCa:=rValorPressaoMaqBar*10197.1621;

(* ---- R_SensorVibracao.prg.st ---- *)
PROGRAM R_SensorVibracao
VAR
	MediaValoresSensorV01: RegistradorMedia;
	MediaValoresSensorV02: RegistradorMedia;
	rValorLeituraSensorVibraV01: REAL;
	rValorLeituraSensorVibraV02: REAL;
	rValorLeituraSensorVibraV01Aux: REAL;
	rValorLeituraSensorVibraV02Aux: REAL;
END_VAR

// Sensor de Vibração Ventilador 01

MediaValoresSensorV01.rDadoEntrada:=INT_TO_REAL(iValorLeituraSensorVibraV01);

MediaValoresSensorV01(rDadoEntrada:= , rDadoSaida=>rValorLeituraSensorVibraV01Aux );

IF	rValorLeituraSensorVibraV01Aux<= 1300 THEN
	rValorLeituraSensorVibraV01:=0;
ELSE
	rValorLeituraSensorVibraV01:=rValorLeituraSensorVibraV01Aux;
END_IF

rValorVibracaoVent01:=((rValorLeituraSensorVibraV01*25)/32767);

// Sensor de Vibração Ventilador 02

MediaValoresSensorV02.rDadoEntrada:=INT_TO_REAL(iValorLeituraSensorVibraV02);

MediaValoresSensorV02(rDadoEntrada:= , rDadoSaida=>rValorLeituraSensorVibraV02Aux );

IF	rValorLeituraSensorVibraV02Aux<= 1300 THEN
	rValorLeituraSensorVibraV02:=0;
ELSE
	rValorLeituraSensorVibraV02:=rValorLeituraSensorVibraV02Aux;
END_IF

rValorVibracaoVent02:=((rValorLeituraSensorVibraV02*25)/32767);

(* ---- S_ElevacaoForno.prg.st ---- *)
PROGRAM S_ElevacaoForno
VAR
	TonSobeForno: TON;
	TonDesceForno: TON;
	AlertaSomCxForno: TimerGeneration;
	AlertaSomCxFornoIn: BOOL;
	AlertaSomCxFornoQ: BOOL;
END_VAR

(*-------------------- Hidraulica -------------------*)
TonSobeForno(IN:=xBtSobeForno , PT:=T#10S , Q=> , ET=> );

xDescendoForno		:=xBtDesceForno;
xSubindoForno		:=xBtSobeForno AND NOT TonSobeForno.Q;

xFechaCaixaForno:=xDescendoForno;
xAbreCaixaForno:=xSubindoForno;
xMotorBombaHidraulica:=xSubindoForno OR xValvulaAvancHidra OR xValvulaRecuoHidra;

IF TonSobeForno.Q THEN
	xBtSobeForno:=FALSE;
END_IF
(*---------------------------------------------------*)

(*------------------- Motorizado --------------------*)

AlertaSomCxFornoIn:=xMotorCaixaFornoLigado;
AlertaSomCxForno(ENABLE:=AlertaSomCxFornoIn , TIMELOW:=T#500mS , TIMEHIGH:=T#500mS , OUT=>AlertaSomCxFornoQ );
xAlertaSomCxForno:=AlertaSomCxFornoQ;

IF rMediaLogicaTemperaturaTotal<=700 THEN
	xBloqAbertCxFornoTemper:=TRUE;
ELSE
	xBloqAbertCxFornoTemper:=FALSE;
END_IF

(* ---- T_Damper.prg.st ---- *)
PROGRAM T_Damper
VAR
	PulsoDamper: PulsoPositivo;
	xPulsoEntradaDamper: BOOL;
	xPulsoSaidaDamper: BOOL;
	xMudancadeDamper: BOOL;
	xValvulaDamperDifusorFino: BOOL;
END_VAR

IF xValvulaDamperDifusor<>xBufferValvulaDamperDifusor THEN
	xMudancadeDamper:=TRUE;
ELSE
	xMudancadeDamper:=FALSE;
END_IF

IF (xMudancadeDamper AND NOT xResfriadorEmCiclo)  THEN
	xPulsoEntradaDamper:=TRUE;
END_IF

PulsoDamper(Entrada:=xPulsoEntradaDamper , SaidaPulsoPo=> xPulsoSaidaDamper);

IF xPulsoSaidaDamper THEN
	xValvulaDamperDifusorFino:=xBufferValvulaDamperDifusor;
END_IF

IF xPulsoEntradaDamper THEN
	xPulsoEntradaDamper:=FALSE;
END_IF

//Saída Damper
xValvulaDamperDifusor:=xValvulaDamperDifusorFino;

(* ---- T_VenezianaDutPass.prg.st ---- *)
PROGRAM T_VenezianaDutPass

IF BtAbreVeneziana THEN
	xValvulaVeneziana:=FALSE;
	BtAbreVeneziana:=FALSE;
END_IF

IF BtFechaVeneziana THEN
	xValvulaVeneziana:=TRUE;
	BtFechaVeneziana:=FALSE;
END_IF

(* ---- T_VenezianaVentInfPass.prg.st ---- *)
PROGRAM T_VenezianaVentInfPass
VAR
	xHabilitaVenezVent01InfPass: BOOL;
	xHabilitaVenezVent02InfPass: BOOL;
	xBloqCmdManVenez: BOOL;
END_VAR

(*// ACIONAMENTO MANUAL

// Habilita/Desabilita Funcionamento Manual
IF xAbreVenezVentPass THEN
	xPassandoTempera:=TRUE;
END_IF
IF xFechVenezVentPass THEN
	xPassandoTempera:=FALSE;
END_IF

IF iVelocidade01Ventilador01<>0 THEN
	xHabilitaVenezVent01InfPass:=TRUE;
ELSE
	xHabilitaVenezVent01InfPass:=FALSE;
END_IF

IF (xHabilitaVenezVent01InfPass OR xHabilitaVenezVent02InfPass) AND xPassandoTempera THEN
	xBloqCmdManVenez:=TRUE;
ELSE
	xBloqCmdManVenez:=FALSE;
END_IF

IF BtAbreVenezVentInfPass AND NOT xBloqCmdManVenez THEN
	xValvulaDamperDifusor:=TRUE;
END_IF
IF BtAbreVenezVentInfPass THEN
	BtAbreVenezVentInfPass:=FALSE;
END_IF

IF BtFechVenezVentInfPass AND NOT xBloqCmdManVenez THEN
	xValvulaDamperDifusor:=FALSE;
END_IF
IF BtFechVenezVentInfPass THEN
	BtFechVenezVentInfPass:=FALSE;
END_IF

// ACIONAMENTO AUTOMATICO

// Habilita Funcionamento Veneziana
IF iVelocidade01Ventilador02<>0 THEN
	xHabilitaVenezVent02InfPass:=TRUE;
ELSE
	xHabilitaVenezVent02InfPass:=FALSE;
END_IF

//Comandos de Abertura e Fechamento
//Abre
IF (xAbreVenezVentPass AND xHabilitaVenezVent02InfPass ) THEN
	xValvulaDamperDifusor:=TRUE;
END_IF
IF xAbreVenezVentPass THEN
	xAbreVenezVentPass:=FALSE;
END_IF

//Fecha
IF xFechaVenezVentPassV01 OR xFechaVenezVentPassV02 OR xFechVenezVentPass THEN
	xValvulaDamperDifusor:=FALSE;
END_IF
IF xFechaVenezVentPassV01 THEN
	xFechaVenezVentPassV01:=FALSE;
END_IF
IF xFechaVenezVentPassV02 THEN
	xFechaVenezVentPassV02:=FALSE;
END_IF
IF xFechVenezVentPass THEN
	xFechVenezVentPass:=FALSE;
END_IF

IF xOperacaoManual THEN
	xPassandoTempera:=FALSE;
	xBloqCmdManVenez:=FALSE;
END_IF

// VELOCIDADE STAND BY VENTILADORES PASSAGEM

IF xHabilitaVenezVent01InfPass THEN
	iVelocidadeStbVent01Pass:=iVelocidadeStbVentilador01;
ELSE
	iVelocidadeStbVent01Pass:=0;
END_IF

IF xHabilitaVenezVent02InfPass THEN
	iVelocidadeStbVent02Pass:=iVelocidadeStbVentilador02;
ELSE
	iVelocidadeStbVent02Pass:=0;
END_IF*)

(* ---- V_VentilacaoPainel.prg.st ---- *)
PROGRAM V_VentilacaoPainel
VAR
	VentiladorPainel: HabilitaDesabilita;
	IniciaTempo: BOOL;
	TOF_Vent: TOF;
	iTolSpTermoPainel: INT;
	iSpTermoparPainelHigh: INT;
	iSpTermoparPainelLow: INT;
	xTermPaiOnOff: BOOL;
END_VAR

//TermoparPainel:=iTemperaturaPirometroPainel;

// Comando Liga Desliga Ventiladores do Painel
// Força Manual

VentiladorPainel(
	Entrada:= xBtLigaVentiPainelManual,
	Entrada02:= ,
	Entrada03:= ,
	Alarme01:= ,
	Alarme02:= ,
	Alarme03:= ,
	StatusSaida=> xLigaVentiPainelManual);

IF xBtLigaVentiPainelManual THEN
	xBtLigaVentiPainelManual:=FALSE;
END_IF

iTolSpTermoPainel:=10;
iSpTermoparPainelHigh:=iSpTermoparPainel+iTolSpTermoPainel;
iSpTermoparPainelLow:=iSpTermoparPainel-iTolSpTermoPainel;

IF Termopar01Painel>=iSpTermoparPainelHigh THEN
	xTermPaiOnOff:=TRUE;
END_IF
IF Termopar01Painel<=iSpTermoparPainelLow THEN
	xTermPaiOnOff:=FALSE;
END_IF

// Automatico
IF xTermPaiOnOff OR xLigaVentiPainelManual THEN
	xVentiladoresPainel:= TRUE;
ELSE
	xVentiladoresPainel:= FALSE;
END_IF

iTemperaturaPainel:=Termopar01Painel;

// Ventiladores dos Reles de Estado Sólidos

	TOF_Vent(IN:=xResistenciasLigadas, PT:= T#600S, Q=>xVentiladoresSsr , ET=> );

(* ---- X_LimpaResfriador02.prg.st ---- *)
PROGRAM X_LimpaResfriador02
VAR
	xResfriador02Aberto: BOOL;
	TonLimpVidroForaPosicao: TON;
	xTonLimpVidroForaPosicaoIn: BOOL;
	xTonLimpVidroForaPosicaoQ: BOOL;
	TonLimpVidroForaPosicaoSom: TP;
	xTonLimpVidroForaPosicaoSomIn: BOOL;
	xTonLimpVidroForaPosicaoSomQ: BOOL;
END_VAR

(*---------------Pré Condição para Funcionamento Limpa Resfriador -------------------*)
(* Resfriador 02 Inferior Totalmente Aberto *)
xResfriador02Aberto:=xSensorAbertoResfriadorInf02 OR xFcMaximoSegResfriadorInf02;

(* Comando do Limpa Vidros Manual *)
xAvancoLimpaResfriador02:=xCHAvancoLimpaResfriador02 AND NOT xFcLimMaxLimpaResfriador02 AND xResfriador02Aberto;
xRecuoLimpaResfriador02:=xCHRecuoLimpaResfriador02 AND NOT xFcLimMinLimpaResfriador02 AND xResfriador02Aberto;

(* Alarme Limpa Vidro Fora de Posição *)

xTonLimpVidroForaPosicaoIn:= NOT xMotorLimpResfr02Ligado AND NOT xFcLimMinLimpaResfriador02;
TonLimpVidroForaPosicao(IN:=xTonLimpVidroForaPosicaoIn , PT:=T#3S , Q=>xTonLimpVidroForaPosicaoQ , ET=> );

IF xTonLimpVidroForaPosicaoQ THEN
	xLimpVidroForaPosicao:=TRUE;
END_IF

(*------------Alerta Sonoro Limpa Vidro fora de Posição --------*)
xTonLimpVidroForaPosicaoSomIn:=xLimpVidroForaPosicao;
TonLimpVidroForaPosicaoSom(IN:= xTonLimpVidroForaPosicaoSomIn, PT:= T#500MS , Q=>xTonLimpVidroForaPosicaoSomQ );

IF xTonLimpVidroForaPosicaoSomQ THEN
	xLimpVidroForaPosicaoSon:=TRUE;
END_IF

IF	bResetAlmGeral THEN
	xLimpVidroForaPosicao:=FALSE;
	xLimpVidroForaPosicaoSon:=FALSE;
END_IF
